Universal Robots PolyScope program: tcp_ip.urp

Program davidz (installation=default directory=/programs/seminar/2526 createdIn=5.11.9.1010452 lastSavedIn=5.11.9.1010452 robotSerialNumber=20185500087)
Calibrated DH parameters: a=[0.000137, -0.413209, -0.387078, 0.000078, -0.000004, 0]; d=[0.162361, 46.755621, 39.772032, -86.394282, 0.099723, 0.099655]; alpha=[1.570462, -0.002125, 0.000722, 1.570578, -1.570334, 0]; deltaTheta=[0, -0.236012, 6.679269, -0.160076, 0, 0]
Robot Program (runOnlyOnce=false)
  Call SubProgram_1
SubProgram -> SubProgram_1
SubProgram SubProgram_1 (keepSynchronizedWithDisk=false)
  Script: open_socket=socket_open("192.168.65.102",50000,"student")
  Loop While (checkContinuously=false) expression=open_socket==False
    Script: open_socket=socket_open("192.168.65.102",50000,"student")
  Popup Message (haltProgram=false message=:) inputType=Text)
  If open_socket==True
    Script: str=socket_read_string("student")
    Loop While (checkContinuously=false) expression=str==""
      Script: str=socket_read_string("student")
      Wait Sleep waitTime=0.01
    Popup Message (haltProgram=false message=rec inputType=Text)
    Script: was_send=socket_send_string("ACK","student")
    Loop While (checkContinuously=false) expression=was_send==False
      Script: was_send=socket_send_string("ACK","student")
      Wait Sleep waitTime=0.01
    Wait Sleep waitTime=0.01
    Popup Message (haltProgram=false message=send inputType=Text)
    Script: read_int=socket_read_binary_integer(1,"student")
    Loop While (checkContinuously=false) expression=read_int[0]==0
      Script: read_int=socket_read_binary_integer(1,"student")
      Wait Sleep waitTime=0.01
    Popup Message (haltProgram=false message=rec inputType=Text)
    Script: was_send=socket_send_int(9,"student")
    Loop While (checkContinuously=false) expression=was_send==False
      Script: was_send=socket_send_int(9,"student")
      Wait Sleep waitTime=0.01
    Wait Sleep waitTime=0.01
    Script: socket_close("student")
    Halt
